PROGRAM PidParameterMenuBindings
VAR
	reactorTemperaturePidParameters : ST_PidParameters;
END_VAR
VAR PERSISTENT
	PbTextField_TextVariable : INT := 9;
	TiTextField_TextVariable : INT := 300;
	TdTextField_TextVariable : INT := 900;
	IterationTimeTextField_TextVariable : INT := 6;
	BiasTextField_TextVariable : INT;
END_VAR


reactorTemperaturePidParameters.PB := PbTextField_TextVariable;
reactorTemperaturePidParameters.Ti := TiTextField_TextVariable;
reactorTemperaturePidParameters.Td := TdTextField_TextVariable;
reactorTemperaturePidParameters.Iterationtime := IterationTimeTextField_TextVariable;
reactorTemperaturePidParameters.Bias := BiasTextField_TextVariable;
ReactorTemperature.pidControllerParameters := reactorTemperaturePidParameters;

END_PROGRAM

(* stored: Version 1.1.0.1, ProductVersion 3.1.4024.9
   POU PidParameterMenuBindings: Id {1a0b8999-6280-4899-bfb0-561a566affd5}, SpecialFunc None *)
